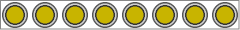
VISUALIZATION v_byte  // 240x30
VAR_IN_OUT
	iNum : INT;
END_VAR
    Lamp1 (0,0 30x30), variable: GVL.stByte.arByte[iNum].Ch[0], style: Lamp-Lamp1-Yellow
    Lamp1 (30,0 30x30), variable: GVL.stByte.arByte[iNum].Ch[1], style: Lamp-Lamp1-Yellow
    Lamp1 (60,0 30x30), variable: GVL.stByte.arByte[iNum].Ch[2], style: Lamp-Lamp1-Yellow
    Lamp1 (90,0 30x30), variable: GVL.stByte.arByte[iNum].Ch[3], style: Lamp-Lamp1-Yellow
    Lamp1 (120,0 30x30), variable: GVL.stByte.arByte[iNum].Ch[4], style: Lamp-Lamp1-Yellow
    Lamp1 (150,0 30x30), variable: GVL.stByte.arByte[iNum].Ch[5], style: Lamp-Lamp1-Yellow
    Lamp1 (180,0 30x30), variable: GVL.stByte.arByte[iNum].Ch[6], style: Lamp-Lamp1-Yellow
    Lamp1 (210,0 30x30), variable: GVL.stByte.arByte[iNum].Ch[7], style: Lamp-Lamp1-Yellow
END_VISUALIZATION

(* stored: Version 1.1.0.1, ProductVersion 3.1.4024.12
   Visu v_byte: Id {b28fd84a-3803-4deb-8308-147e0adde3ed} *)
